FUNCTION_BLOCK System_TaskInfo
VAR_INPUT
	
END_VAR
VAR_OUTPUT
	// Object ID of the task reference, from which the PLC program is called.
	ObjId: UDINT;
	// Set task cycle time in multiples of 100 ns
	CycleTime: UDINT;
	// Set task priority
	Priority: UINT;
	// ADS port of the task
	AdsPort: UINT;
	(* 
	Cycle counter
	Please note that the cycle counter refers to the actual system task 
	and not to the task reference of the PLC project. The background to 
	this is that several PLC projects or other TcCOM modules can share 
	a task and these modules can thus access the same cycle counter. 
	As a result, the cycle counter is reset during a TwinCAT restart in 
	RUN mode (and not when resetting the PLC project). *)
	CycleCount: UDINT;
	// Distributed Clock System Time. It remains constant for a task runtime.
	DcTaskTime: LINT;
	// Cycle time required for the last cycle in multiples of 100 ns
	LastExecTime: UDINT;
	// During the first PLC task cycle, this variable has the value TRUE.
	FirstCycle: BOOL;
	(* 
	This variable indicates whether the set task cycle time was exceeded.
	The value of the CycleTimeExceeded variable is updated in each cycle. 
	The variable is set to 0 if the previous cycle has been completed 
	within its intended timeframe, otherwise to 1. *)
	CycleTimeExceeded: BOOL;
	(* 
	This variable has the value TRUE if the origin of the current call 
	is declared with the attribute 'TcCallAfterOutputUpdate'. *)
	InCallAfterOutputUpdate: BOOL;
	(* This variable has the value TRUE if the real-time limit is 
	exceeded on a mixed core (Windows + real-time on one core). In this 
	case the value TRUE refers to the core on which the corresponding 
	task is running. *)
	RTViolation: BOOL;
	// Name of the task reference object in the PLC project (e.g. 'MyPlcProject_PlcTaskRef')
	TaskName: STRING(63);
END_VAR
VAR
	
	_ThisTaskInfo: PlcTaskSystemInfo;
	_AllTaskInfo : ARRAY[0..10] OF PlcTaskSystemInfo;
	index : UDINT;
	TaskCount : UDINT;
	TaskIndex : DINT ;
	
	
END_VAR

TaskCount := _AppInfo.TaskCnt;
FOR index := 1 TO LIMIT(1,TaskCount,10)  DO
	_AllTaskInfo[index] := _TaskInfo[index];
END_FOR
TaskIndex := GETCURTASKINDEXEX();
_ThisTaskInfo := _AllTaskInfo[TaskIndex];

_ThisTaskInfo := _TaskInfo[TaskIndex];
ObjId := _ThisTaskInfo.ObjId; 
CycleTime := _ThisTaskInfo.CycleTime;
Priority := _ThisTaskInfo.Priority;
AdsPort := _ThisTaskInfo.AdsPort;
CycleCount := _ThisTaskInfo.CycleCount;
DcTaskTime := _ThisTaskInfo.DcTaskTime;
LastExecTime := _ThisTaskInfo.LastExecTime;
FirstCycle := _ThisTaskInfo.FirstCycle;
CycleTimeExceeded := _ThisTaskInfo.CycleTimeExceeded;
InCallAfterOutputUpdate := _ThisTaskInfo.InCallAfterOutputUpdate;
RTViolation := _ThisTaskInfo.RTViolation;

TaskName := _ThisTaskInfo.TaskName;

METHOD getCurrentTaskInfo : REFERENCE TO PlcTaskSystemInfo
VAR_INPUT
END_VAR
getCurrentTaskInfo REF= _ThisTaskInfo;
END_METHOD

METHOD getTaskCount : UDINT
VAR_INPUT
END_VAR
getTaskCount := _AppInfo.TaskCnt;
END_METHOD

METHOD getTaskFirstIndex : UDINT
VAR_INPUT
END_VAR
getTaskFirstIndex := 1;
END_METHOD

METHOD getTaskInfoByIndex : REFERENCE TO PlcTaskSystemInfo
VAR_INPUT
	Index : UDINT;
END_VAR
IF Index >= 1 AND index <= 10 THEN
	getTaskInfoByIndex REF= _AllTaskInfo[Index];
ELSE
	getTaskInfoByIndex REF= _AllTaskInfo[0];
END_IF
END_METHOD

END_FUNCTION_BLOCK

(* stored: Version 1.1.0.1, ProductVersion 3.1.4024.12
   POU System_TaskInfo: Id {71654526-854d-4355-b3ed-2a3225024daa}, SpecialFunc None
   Method getCurrentTaskInfo: Id {9b165994-b4dc-4657-87c4-3050d2c4a124}
   Method getTaskCount: Id {93676102-8b09-4b36-8f8b-f0de6a6f820a}
   Method getTaskFirstIndex: Id {401ea817-bd30-421f-8676-b30a16f9ceae}
   Method getTaskInfoByIndex: Id {a8c1a45a-45ea-4f4b-b3da-74508aad500f} *)
